// TwinCAT 3 PLC project ExtruderControl
// ProgramVersion: 3.1.4023.0
// libraries:
//   Tc2_MC2, * (Beckhoff Automation GmbH)
//   Tc2_Standard, * (Beckhoff Automation GmbH)
//   Tc2_System, * (Beckhoff Automation GmbH)
//   Tc3_Module, * (Beckhoff Automation GmbH)
//   VisuDialogs, * (System)
// project tree:
//   DUTs/ Modes.TcDUT
//   / GlobalTextList.TcGTLO, PlcTask.TcTTO, Visualization Manager.TcVMO (not stored)
//   GVLs/ GVL.TcGVL, HMI.TcGVL, IO.TcGVL, MC.TcGVL
//   POUs/ AutoExtrusion.TcPOU, MAIN.TcPOU, Motion.TcPOU, OperatingModes.TcPOU
//   POUs/VISUCode/ VisuLogic.TcPOU (not stored)
//   VISUs/ MainHMI.TcVIS
// real-time tasks:
//   TASK PlcTask: cycle T#10ms, priority 20, ADS port 350
// motion (NC):
//   TASK NC-Task Extruder SAF: cycle T#2ms, priority 4, ADS port 501
//   TASK NC-Task Extruder SVB: cycle T#10ms, priority 8, ADS port 511
//   AXIS ExtruderAxis (id 1)
//     OtherSettings: AllowMotionCmdToSlave=true
//     encoder EncType=1
//     drive DrvType=5
//       Analog: TorqueSetpointScale=10, ScaleFactorActTorque=0.1
//     controller CtrType=1
//       CtrPara: PriorControlFactor=1
//         Observer: BandWidth=20
// variable links:
//   ExtruderControl/ExtruderControl Instance <-> NC-Task Extruder SAF/Axes/ExtruderAxis
//     PlcTask Inputs/MC.Extruder.NcToPlc <-> Outputs/ToPlc
//     PlcTask Outputs/MC.Extruder.PlcToNc <-> Inputs/FromPlc

CONFIGURATION ExtruderControl
    RESOURCE PLC ON TwinCAT3
        TASK PlcTask(INTERVAL := T#10ms, PRIORITY := 20);
        PROGRAM MAIN WITH PlcTask : MAIN;
    END_RESOURCE
END_CONFIGURATION

// ---- DUTs/Modes.TcDUT
{attribute 'qualified_only'}
{attribute 'strict'}
TYPE Modes :
(
	STOP_EM := 0,
	STOP_OP := 1,
	AUTO := 2,
	MAN := 3
);
END_TYPE

// ---- GVLs/GVL.TcGVL
{attribute 'qualified_only'}
VAR_GLOBAL
	
	Mode: Modes;
END_VAR

// ---- GVLs/HMI.TcGVL
{attribute 'qualified_only'}
VAR_GLOBAL
	

	// Modes control
	Bt_Run: BOOL;
	Bt_Stop: BOOL;
	Sel_ManAuto: BOOL := TRUE;
	Bt_EmStop: BOOL;
	Bt_Rearm:BOOL;
	Bt_Front: BOOL;
	Bt_Back:BOOL;
	
	//Process Control
	Bt_StartCycle:BOOL;
	Tb_Vel:LREAL;
	Tb_TempL:LREAL;
	Tb_TempU:LREAL;
	Tb_Temp:LREAL;
	
END_VAR

// ---- GVLs/IO.TcGVL
{attribute 'qualified_only'}
VAR_GLOBAL
	
	// Heater outputs
	O_HeaterT AT %Q*:BOOL;
	O_HeaterB AT %Q*:BOOL;
	
	// RTD Sensors (PT100)
	I_TermT AT %I*:LREAL;
	I_TermB AT %I*:LREAL;
	
END_VAR

// ---- GVLs/MC.TcGVL
{attribute 'qualified_only'}
VAR_GLOBAL
	// Axis ref
	Extruder: AXIS_REF;
	
	// Orders
	En_Power:BOOL;
	Exec_Stop:BOOL;
	Exec_Velocity:BOOL;
	Exec_Relative:BOOL;
	
	// Motion variables
	Override:LREAL := 100;
	TargetVel:LREAL;
	TargetPosRel:LREAL;
	TargetDirection:MC_Direction;
END_VAR

VAR_GLOBAL CONSTANT
	// Motion constants
	StdVel:LREAL:= 100;
	StdAcc:LREAL:= 1000;
	StdDecc:LREAL:= 1000;
END_VAR

// ---- POUs/MAIN.TcPOU
PROGRAM MAIN
VAR
	
END_VAR

Motion.InitMotion();


OperatingModes();
VisuLogic();
Motion();

END_PROGRAM

// ---- POUs/Motion.TcPOU
PROGRAM Motion
VAR
	FB_Power: MC_Power;
	FB_Stop: MC_Stop;
	FB_Velocity: MC_MoveVelocity;
	FB_Relative: MC_MoveRelative;
	FB_ReadStatus: MC_ReadStatus;

	
END_VAR

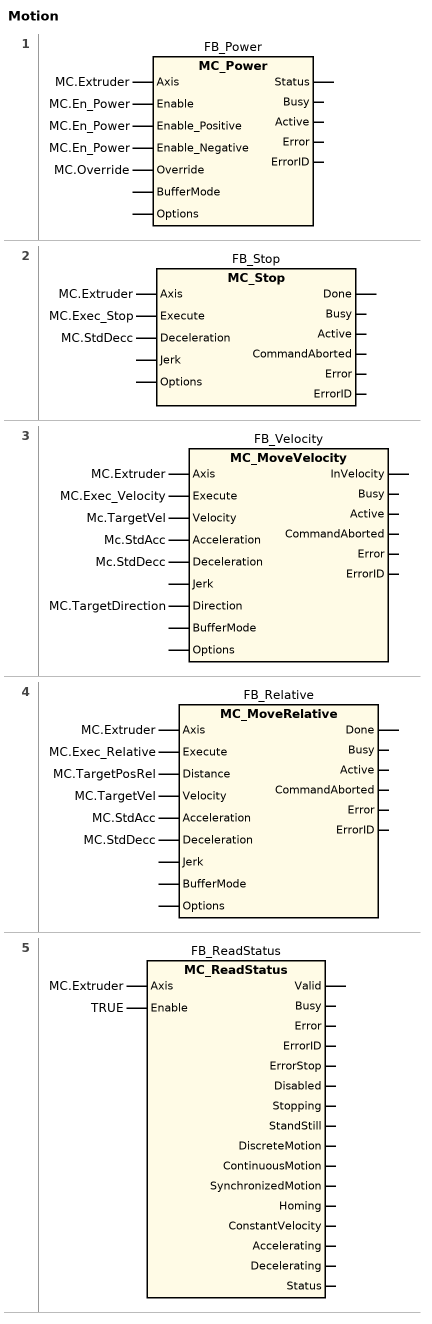
// NETWORK 1
FB_Power(
    Axis := MC.Extruder,
    Enable := MC.En_Power,
    Enable_Positive := MC.En_Power,
    Enable_Negative := MC.En_Power,
    Override := MC.Override); // MC_Power

// NETWORK 2
FB_Stop(Axis := MC.Extruder, Execute := MC.Exec_Stop, Deceleration := MC.StdDecc); // MC_Stop

// NETWORK 3
FB_Velocity(
    Axis := MC.Extruder,
    Execute := MC.Exec_Velocity,
    Velocity := Mc.TargetVel,
    Acceleration := Mc.StdAcc,
    Deceleration := Mc.StdDecc,
    Direction := MC.TargetDirection); // MC_MoveVelocity

// NETWORK 4
FB_Relative(
    Axis := MC.Extruder,
    Execute := MC.Exec_Relative,
    Distance := MC.TargetPosRel,
    Velocity := MC.TargetVel,
    Acceleration := MC.StdAcc,
    Deceleration := MC.StdDecc); // MC_MoveRelative

// NETWORK 5
FB_ReadStatus(Axis := MC.Extruder, Enable := TRUE); // MC_ReadStatus

ACTION InitMotion:
Mc.En_Power := FALSE;
MC.Exec_Relative := FALSE;
MC.Exec_Stop := FALSE;
MC.Exec_Velocity := FALSE;
END_ACTION

END_PROGRAM

// ---- POUs/OperatingModes.TcPOU
PROGRAM OperatingModes
VAR
	AuxStopping:Modes;
END_VAR

CASE GVL.Mode OF
	
	// Emergency stop
	Modes.STOP_EM:
		IF HMI.Bt_Rearm THEN
			gvl.Mode := modes.STOP_OP;
		END_IF
	
	// Operative stop
	Modes.STOP_OP:
		IF HMI.Bt_EmStop THEN
			GVL.Mode := Modes.STOP_EM;
		END_IF
		IF HMI.Bt_Run AND HMI.Sel_ManAuto THEN
			GVL.Mode := Modes.AUTO;
		END_IF
		IF NOT HMI.Sel_ManAuto THEN
			GVL.Mode := Modes.MAN;
		END_IF
		
	// Automatic
	Modes.AUTO:
		IF HMI.Bt_EmStop THEN
			GVL.Mode := Modes.STOP_EM;
		END_IF
		IF NOT HMI.Sel_ManAuto THEN
			GVL.Mode := Modes.MAN;
		END_IF
		IF HMI.Bt_Stop THEN
			GVL.Mode := Modes.Stopping;
			AuxStopping := Modes.STOP_OP;
		END_IF
		
	// Manual
	Modes.MAN:
		IF HMI.Bt_EmStop THEN
			GVL.Mode := Modes.STOP_EM;
		END_IF
		IF HMi.Sel_ManAuto THEN
			GVL.Mode := Modes.STOP_OP;
		END_IF	
		
	// Stopping
	Modes.Stopping:
		MC.Exec_Stop:= TRUE;
		IF Motion.FB_Stop.Done THEN
			GVL.Mode := AuxStopping;
		END_IF
END_CASE

// Axis Power when not in stop
IF GVL.Mode <> Modes.STOP_EM THEN
	MC.En_Power := TRUE;
END_IF

END_PROGRAM

// ---- POUs/AutoExtrusion.TcPOU
PROGRAM AutoExtrusion
VAR
END_VAR

END_PROGRAM

// ---- GlobalTextList.TcGTLO
TEXTLIST GlobalTextList
  403 = '%s'
  734 = '%s ºC'
  600 = 'Auto             Manual'
  864 = 'Auto        Manual'
  794 = 'Automatic' | Galician: 'Automático'
  481 = 'Bottom Heater' | Galician: 'Calefactor inferior'
  766 = 'Emergency' | Galician: 'Emerxencia'
  130 = 'Error' | Galician: 'Erro'
  673 = 'Extruder' | Galician: 'Extrusor'
  542 = 'Manual' | Galician: 'Manual'
  668 = 'Modo: %s'
  653 = 'Moving' | Galician: 'Movendose'
  275 = 'Operating modes' | Galician: 'Modos de operación'
  139 = 'Power' | Galician: 'Potencia'
  586 = 'Rearm' | Galician: 'Rearme'
  688 = 'Start' | Galician: 'Inicio'
  765 = 'Start Cycle' | Galician: 'Iniciar ciclo'
  988 = 'Status' | Galician: 'Estado'
  954 = 'Stop' | Galician: 'Parada'
  385 = 'STOP' | Galician: 'Paro'
  524 = 'Temperature' | Galician: 'Temperatura'
  559 = 'Top Heater' | Galician: 'Calefactor superior'
  367 = 'Velocity' | Galician: 'Velocidade'
END_TEXTLIST

// ---- VISUs/MainHMI.TcVIS
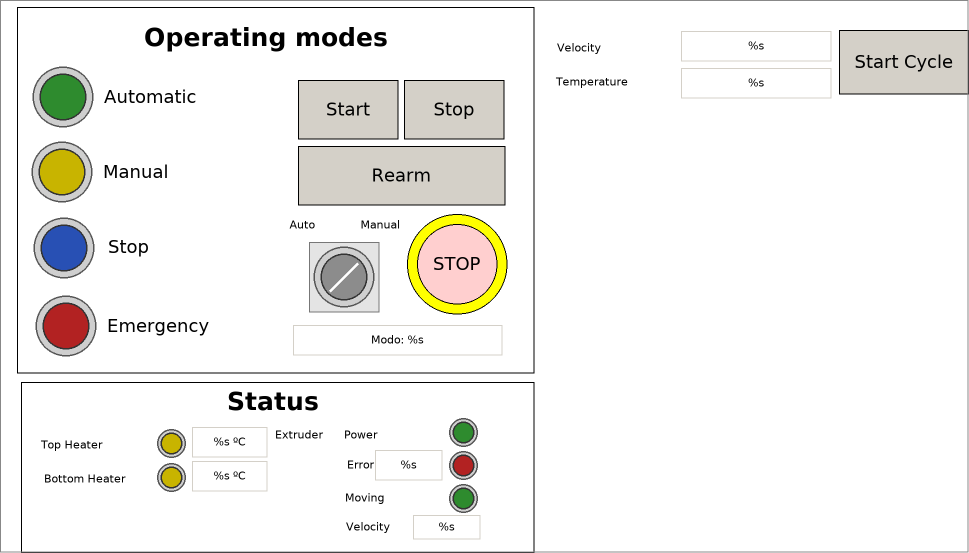
VISUALIZATION MainHMI  // 969x553
    RoundedRectangle (21,382 513x171)
    RoundedRectangle (17,7 517x366)
    Lamp1 (28,62 70x70), variable: VisuLogic.L_Run, style: Lamp-Lamp1-Green
    Label (101,82 118x30), "Automatic"
    Label (100,157 119x30), "Manual"
    Lamp1 (27,137 70x70), variable: VisuLogic.L_Manual, style: Lamp-Lamp1-Yellow
    Label (105,232 114x30), "Stop"
    Lamp1 (29,213 70x70), variable: VisuLogic.L_StopOP, style: Lamp-Lamp1-Blue
    Label (104,311 115x30), "Emergency"
    Lamp1 (31,291 70x70), variable: VisuLogic.L_StopEM, style: Lamp-Lamp1-Red
    Rectangle (298,80 100x59), "Start"
        tap HMI.Bt_Run
    Rectangle (404,80 100x59), "Stop"
        tap HMI.Bt_Stop
    Rectangle (298,146 207x59), "Rearm"
        tap HMI.Bt_Rearm
    Ellipse (407,214 100x100)
    Ellipse (417,224 80x80), "STOP"
        toggle HMI.Bt_EmStop
    RotarySwitch (309,242 70x70), variable: HMI.Sel_ManAuto, behaviour: TOGGLE, style: Switch-RotarySwitch-Gray
    Label (284,210 122x30), "Auto Manual"
    Label (124,22 284x30), "Operating modes"
    Textfield (681,31 150x30), "%s", text variable: HMI.Tb_Vel
        OnMouseDown: write HMI.Tb_Vel via VisuDialogs.Numpad
    Label (554,33 120x30), "Velocity"
    Rectangle (839,30 130x64), "Start Cycle"
        tap HMI.Bt_StartCycle
    Label (553,67 120x30), "Temperature"
    Textfield (681,68 150x30), "%s", text variable: HMI.Tb_Temp
        OnMouseDown: write HMI.Tb_Temp via VisuDialogs.Keypad
    Label (131,386 284x30), "Status"
    Lamp1 (155,427 33x33), variable: IO.O_HeaterT, style: Lamp-Lamp1-Yellow
    Lamp1 (155,461 33x33), variable: IO.O_HeaterB, style: Lamp-Lamp1-Yellow
    Label (38,430 150x30), "Top Heater"
    Label (41,464 150x30), "Bottom Heater"
    Textfield (192,427 75x30), "%s ºC", text variable: IO.I_TermT
    Textfield (192,461 75x30), "%s ºC", text variable: IO.I_TermB
    Label (272,420 57x30), "Extruder"
    Lamp1 (447,449 33x33), variable: MC.Extruder.Status.Error, style: Lamp-Lamp1-Red
    Lamp1 (447,416 33x33), variable: Motion.FB_Power.Status, style: Lamp-Lamp1-Green
    Label (341,420 57x30), "Power"
    Label (344,450 57x30), "Error"
    Textfield (375,450 67x30), "%s", text variable: MC.Extruder.Status.ErrorID
    Lamp1 (447,482 33x33), variable: MC.Extruder.Status.Moving, style: Lamp-Lamp1-Green
    Label (342,483 103x30), "Moving"
    Label (343,512 57x30), "Velocity"
    Textfield (413,515 67x24), "%s", text variable: MC.Extruder.NcToPlc.ActVelo
    Textfield (293,325 209x30), "Modo: %s", text variable: GVL.Mode
END_VISUALIZATION
